ADAPTER IAS_Skill
  (* Standard: 61499-1 *)
  (* Version 0.0, 2008-04-22, GE, 4DIAC-Consortium *)
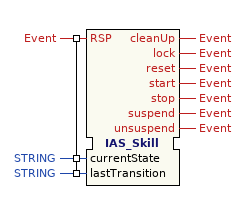
  EVENT_INPUT
    RSP WITH currentState, lastTransition;
  END_EVENT
  EVENT_OUTPUT
    cleanUp;
    lock;
    reset;
    start;
    stop;
    suspend;
    unsuspend;
  END_EVENT
  VAR_INPUT
    currentState : STRING;
    lastTransition : STRING;
  END_VAR
  SERVICE SOCKET/PLUG
    SEQUENCE request_confirm
      SOCKET.REQ(REQD) -> PLUG.REQ(REQD);
      PLUG.CNF(CNFD) -> SOCKET.CNF(CNFD);
    END_SEQUENCE
    SEQUENCE indication_response
      PLUG.IND(INDD) -> SOCKET.IND(INDD);
      SOCKET.RSP(RSPD) -> PLUG.RSP(RSPD);
    END_SEQUENCE
  END_SERVICE
END_ADAPTER
